PROGRAM MAIN
VAR	
	fbToggle : FB_Toggle;
	fbTimerPulse : FB_TimerPulse;
	bStart : BOOL;
	fbTrigger : FB_Triggers;
END_VAR


IF bStart THEN
	fbTimerPulse();
	//fbToggle();
	//fbTrigger();
END_IF

END_PROGRAM

(* stored: Version 1.1.0.1, ProductVersion 3.1.4024.16
   POU MAIN: Id {12b2fffa-9e32-409e-9fc5-570eed32ce65}, SpecialFunc None *)
